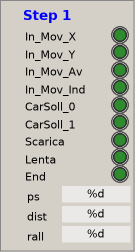
VISUALIZATION Programma  // 135x252
    Label (22,22 100x30), "In_Mov_X"
    Label (22,40 113x30), "In_Mov_Y"
    Lamp1 (110,25 20x20), variable: fbClassAsrv.sAsrv.ASRV_MIS.Step_PC[1].Comandi.In_Mov_X, style: Lamp-Lamp1-Green
    Lamp1 (110,42 20x20), variable: sLastStep.Comandi.In_Mov_Y, style: Lamp-Lamp1-Green
    Label (22,57 113x30), "In_Mov_Av"
    Label (22,75 113x30), "In_Mov_Ind"
    Lamp1 (110,60 20x20), variable: sLastStep.Comandi.In_Mov_Av, style: Lamp-Lamp1-Green
    Lamp1 (110,77 20x20), variable: sLastStep.Comandi.In_Mov_Ind, style: Lamp-Lamp1-Green
    Label (24,202 40x30), "dist"
    Label (24,222 40x30), "rall"
    Textfield (61,205 70x18), "%d", text variable: sLastStep.dist
    Textfield (61,225 70x18), "%d", text variable: sLastStep.rall
    Label (24,182 40x30), "ps"
    Textfield (61,185 70x18), "%d", text variable: sLastStep.ps
    Label (22,92 113x30), "CarSoll_0"
    Label (22,110 113x30), "CarSoll_1"
    Lamp1 (110,95 20x20), variable: sLastStep.Comandi.CarSoll_0, style: Lamp-Lamp1-Green
    Lamp1 (110,112 20x20), variable: sLastStep.Comandi.CarSoll_1, style: Lamp-Lamp1-Green
    Label (22,127 113x30), "Scarica"
    Label (22,145 113x30), "Lenta"
    Lamp1 (110,130 20x20), variable: sLastStep.Comandi.Scarica, style: Lamp-Lamp1-Green
    Lamp1 (110,147 20x20), variable: sLastStep.Comandi.Lenta, style: Lamp-Lamp1-Green
    Label (22,162 113x30), "End"
    Lamp1 (110,164 20x20), variable: sLastStep.Comandi.End, style: Lamp-Lamp1-Green
    Label (20,4 100x23), "Step 1"
END_VISUALIZATION

(* stored: Version 1.1.0.1, ProductVersion 3.1.4024.11
   Visu Programma: Id {48f814e0-f07f-4043-b73e-51582d8e4744} *)
